Staubli VAL3: remGetHere.pgx

program remGetHere(string& sReturn[] (dimensions=1))
begin
  // Return current position in Cartesian coordinates
  //
  logMsg("call remGetHere")
  call remCalcHere()
  sReturn="GETPOS"
  sReturn=sReturn+" "+toString(sNumConv,nXHere)
  sReturn=sReturn+" "+toString(sNumConv,nYHere)
  sReturn=sReturn+" "+toString(sNumConv,nZHere)
  sReturn=sReturn+" "+toString(sNumConv,nRXHere)
  sReturn=sReturn+" "+toString(sNumConv,nRYHere)
  sReturn=sReturn+" "+toString(sNumConv,nRZHere)
end
